INTERFACE I_FallibleWord


PROPERTY Error : BOOL
GET
END_GET
END_PROPERTY


PROPERTY Value : WORD
GET
END_GET
END_PROPERTY

END_INTERFACE

(* stored: Version 1.1.0.1
   Itf I_FallibleWord: Id {a1b2c3d4-0001-4001-8001-000000000001}
   Property Error: Id {a1b2c3d4-0001-4001-8001-000000000002}
   Get Get: Id {a1b2c3d4-0001-4001-8001-000000000003}
   Property Value: Id {a1b2c3d4-0001-4001-8001-000000000004}
   Get Get: Id {a1b2c3d4-0001-4001-8001-000000000005} *)
